PROGRAM PRG_RetiradaAlmacen
VAR
END_VAR

END_PROGRAM

(* stored: Version 1.1.0.1, ProductVersion 3.1.4024.12
   POU PRG_RetiradaAlmacen: Id {3c072e24-b3a5-4d0d-b488-8a342df77b82}, SpecialFunc None *)
